{attribute addProperty BoxType "IL2301-B110-0016"}
{attribute addProperty Id "Term_21KL_5BCCED4C00Term_392_Ix1000KL_9BB4615400"}
{attribute addProperty CRC "417716904"}
{attribute addProperty SizeInBites "0"}
{attribute addProperty SizeInBytes "0"}
TYPE A_0021_IL2301_B110_0016_18E5DAA8 EXTENDS IL2301_4487A81F :
STRUCT
	{attribute addProperty Name "Term_21"}
	Term_21 : KL_5BCCED4C;
	{attribute addProperty Name "Term_392_Ix1000"}
	Term_392_Ix1000 : KL_9BB46154;
END_STRUCT
END_TYPE

(* stored: Version 1.2.0.0, ProductVersion 3.1.4024.9
   DUT A_0021_IL2301_B110_0016_18E5DAA8: Id {201ac0b7-5507-45a4-8139-4f2a33c799f1} *)
